(* Logix 5000 project; controller BTS01 vendor 1 type 14 code 217 rev 32.14; software revision 32.04; part 8 of 15 *)
(* tags used below, declared in another part *)
   Alarm_Active : DINT;
   Alarm_TMR : TIMER[17,32];
   ALM_ENABLE : DINT[25];
   HMI_Global_Alarm_Ack_PB : BOOL;
   HMIAlarms : DINT[25];   // Alarm Trigger Array
   HMIAlarmsMsg : STRING64[17,32];   // Alarm Descriptions to Match Alarm Trigger Array
(* Alarm, continued *)

ROUTINE Alarm_07   (* ladder *)
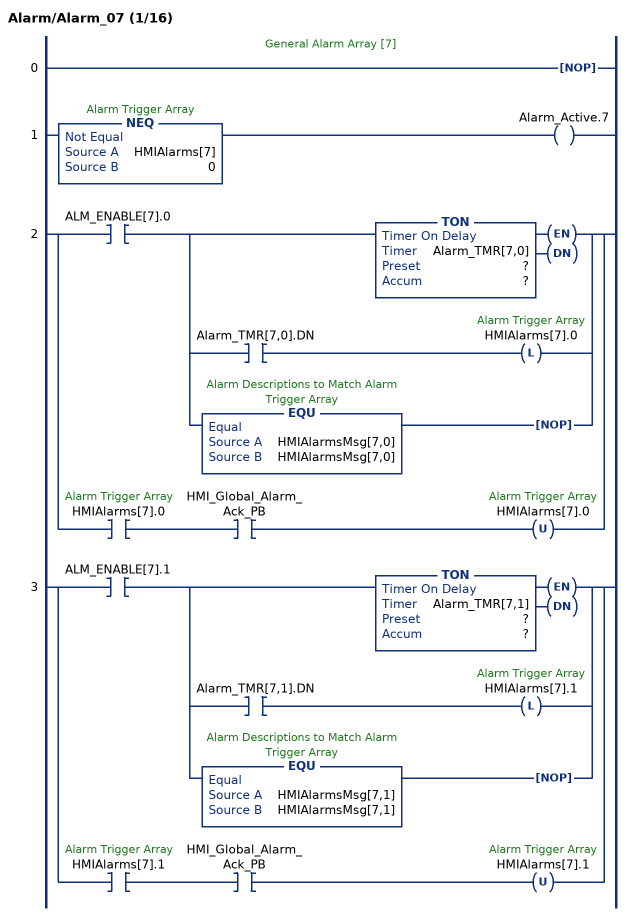
   // General Alarm Array [7]
   0: NOP();
   1: NEQ(HMIAlarms[7],0)OTE(Alarm_Active.7);
   2: [XIC(ALM_ENABLE[7].0) [TON(Alarm_TMR[7,0],?,?) ,XIC(Alarm_TMR[7,0].DN) OTL(HMIAlarms[7].0) ,EQU(HMIAlarmsMsg[7,0],HMIAlarmsMsg[7,0]) NOP() ] ,XIC(HMIAlarms[7].0) XIC(HMI_Global_Alarm_Ack_PB) OTU(HMIAlarms[7].0) ];
   3: [XIC(ALM_ENABLE[7].1) [TON(Alarm_TMR[7,1],?,?) ,XIC(Alarm_TMR[7,1].DN) OTL(HMIAlarms[7].1) ,EQU(HMIAlarmsMsg[7,1],HMIAlarmsMsg[7,1]) NOP() ] ,XIC(HMIAlarms[7].1) XIC(HMI_Global_Alarm_Ack_PB) OTU(HMIAlarms[7].1) ];
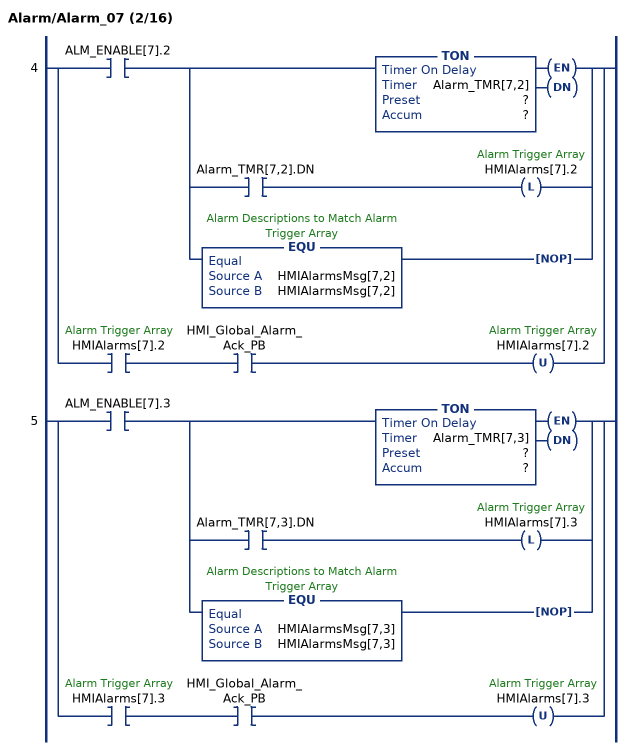
   4: [XIC(ALM_ENABLE[7].2) [TON(Alarm_TMR[7,2],?,?) ,XIC(Alarm_TMR[7,2].DN) OTL(HMIAlarms[7].2) ,EQU(HMIAlarmsMsg[7,2],HMIAlarmsMsg[7,2]) NOP() ] ,XIC(HMIAlarms[7].2) XIC(HMI_Global_Alarm_Ack_PB) OTU(HMIAlarms[7].2) ];
   5: [XIC(ALM_ENABLE[7].3) [TON(Alarm_TMR[7,3],?,?) ,XIC(Alarm_TMR[7,3].DN) OTL(HMIAlarms[7].3) ,EQU(HMIAlarmsMsg[7,3],HMIAlarmsMsg[7,3]) NOP() ] ,XIC(HMIAlarms[7].3) XIC(HMI_Global_Alarm_Ack_PB) OTU(HMIAlarms[7].3) ];
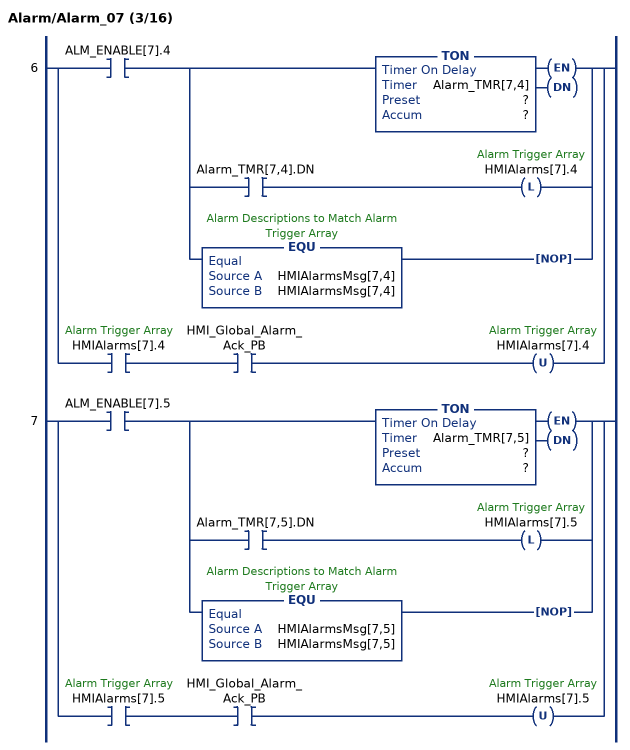
   6: [XIC(ALM_ENABLE[7].4) [TON(Alarm_TMR[7,4],?,?) ,XIC(Alarm_TMR[7,4].DN) OTL(HMIAlarms[7].4) ,EQU(HMIAlarmsMsg[7,4],HMIAlarmsMsg[7,4]) NOP() ] ,XIC(HMIAlarms[7].4) XIC(HMI_Global_Alarm_Ack_PB) OTU(HMIAlarms[7].4) ];
   7: [XIC(ALM_ENABLE[7].5) [TON(Alarm_TMR[7,5],?,?) ,XIC(Alarm_TMR[7,5].DN) OTL(HMIAlarms[7].5) ,EQU(HMIAlarmsMsg[7,5],HMIAlarmsMsg[7,5]) NOP() ] ,XIC(HMIAlarms[7].5) XIC(HMI_Global_Alarm_Ack_PB) OTU(HMIAlarms[7].5) ];
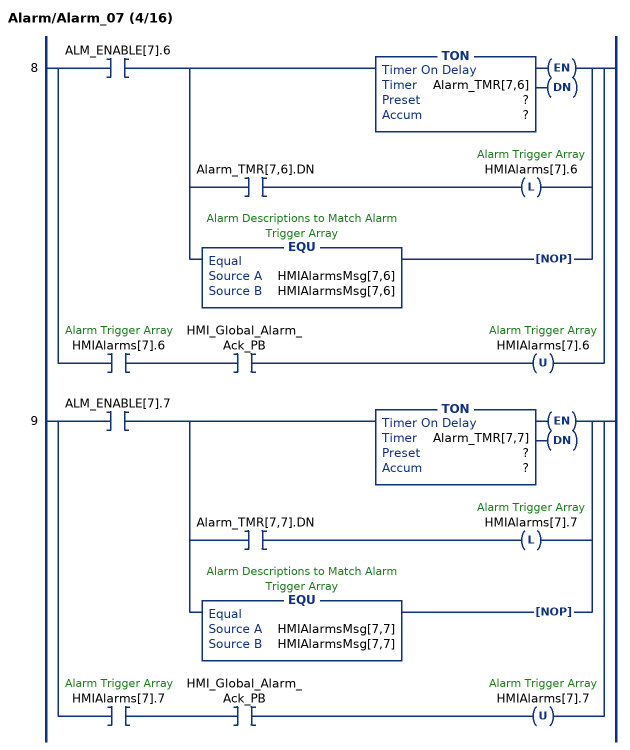
   8: [XIC(ALM_ENABLE[7].6) [TON(Alarm_TMR[7,6],?,?) ,XIC(Alarm_TMR[7,6].DN) OTL(HMIAlarms[7].6) ,EQU(HMIAlarmsMsg[7,6],HMIAlarmsMsg[7,6]) NOP() ] ,XIC(HMIAlarms[7].6) XIC(HMI_Global_Alarm_Ack_PB) OTU(HMIAlarms[7].6) ];
   9: [XIC(ALM_ENABLE[7].7) [TON(Alarm_TMR[7,7],?,?) ,XIC(Alarm_TMR[7,7].DN) OTL(HMIAlarms[7].7) ,EQU(HMIAlarmsMsg[7,7],HMIAlarmsMsg[7,7]) NOP() ] ,XIC(HMIAlarms[7].7) XIC(HMI_Global_Alarm_Ack_PB) OTU(HMIAlarms[7].7) ];
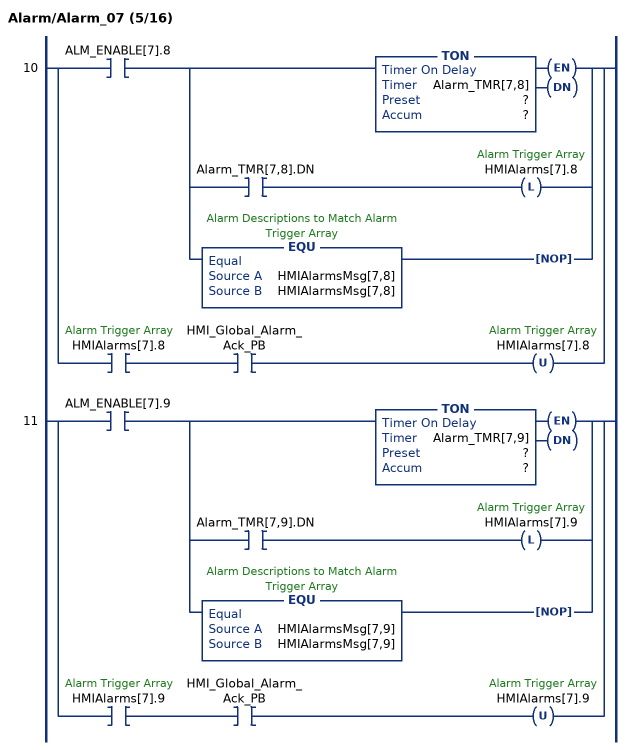
   10: [XIC(ALM_ENABLE[7].8) [TON(Alarm_TMR[7,8],?,?) ,XIC(Alarm_TMR[7,8].DN) OTL(HMIAlarms[7].8) ,EQU(HMIAlarmsMsg[7,8],HMIAlarmsMsg[7,8]) NOP() ] ,XIC(HMIAlarms[7].8) XIC(HMI_Global_Alarm_Ack_PB) OTU(HMIAlarms[7].8) ];
   11: [XIC(ALM_ENABLE[7].9) [TON(Alarm_TMR[7,9],?,?) ,XIC(Alarm_TMR[7,9].DN) OTL(HMIAlarms[7].9) ,EQU(HMIAlarmsMsg[7,9],HMIAlarmsMsg[7,9]) NOP() ] ,XIC(HMIAlarms[7].9) XIC(HMI_Global_Alarm_Ack_PB) OTU(HMIAlarms[7].9) ];
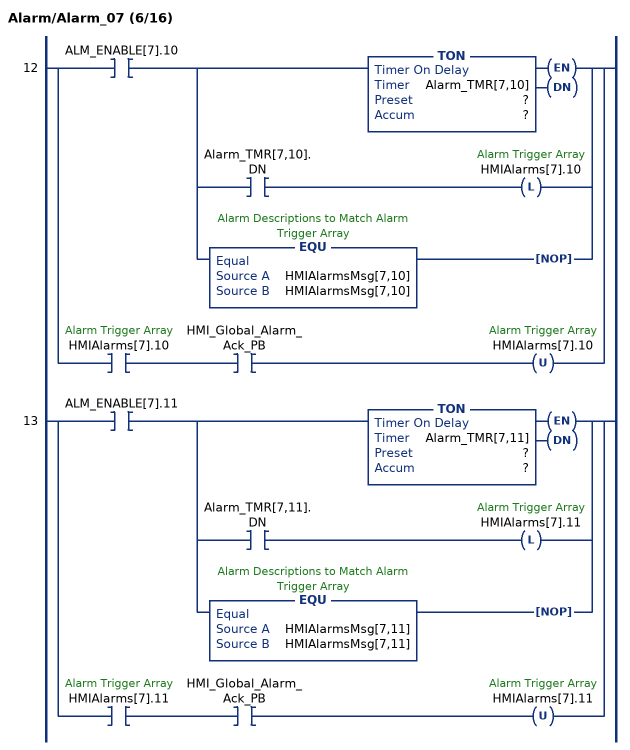
   12: [XIC(ALM_ENABLE[7].10) [TON(Alarm_TMR[7,10],?,?) ,XIC(Alarm_TMR[7,10].DN) OTL(HMIAlarms[7].10) ,EQU(HMIAlarmsMsg[7,10],HMIAlarmsMsg[7,10]) NOP() ] ,XIC(HMIAlarms[7].10) XIC(HMI_Global_Alarm_Ack_PB) OTU(HMIAlarms[7].10) ];
   13: [XIC(ALM_ENABLE[7].11) [TON(Alarm_TMR[7,11],?,?) ,XIC(Alarm_TMR[7,11].DN) OTL(HMIAlarms[7].11) ,EQU(HMIAlarmsMsg[7,11],HMIAlarmsMsg[7,11]) NOP() ] ,XIC(HMIAlarms[7].11) XIC(HMI_Global_Alarm_Ack_PB) OTU(HMIAlarms[7].11) ];
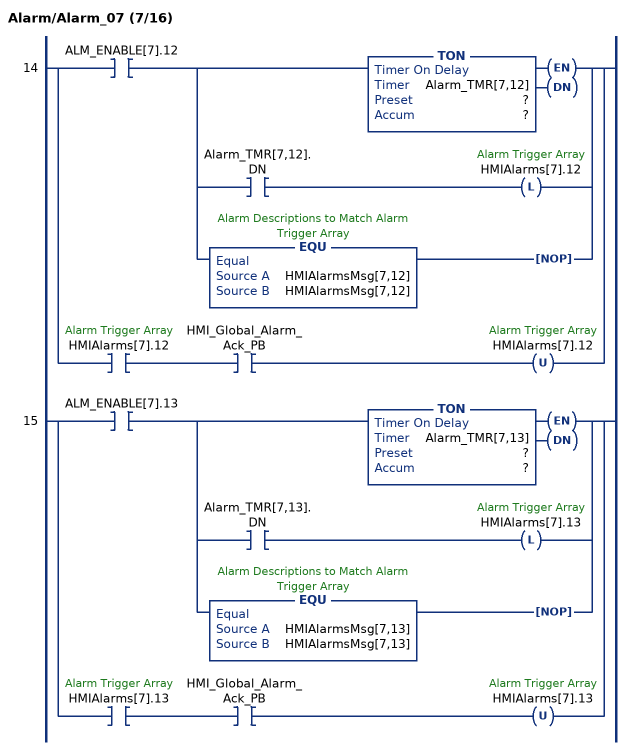
   14: [XIC(ALM_ENABLE[7].12) [TON(Alarm_TMR[7,12],?,?) ,XIC(Alarm_TMR[7,12].DN) OTL(HMIAlarms[7].12) ,EQU(HMIAlarmsMsg[7,12],HMIAlarmsMsg[7,12]) NOP() ] ,XIC(HMIAlarms[7].12) XIC(HMI_Global_Alarm_Ack_PB) OTU(HMIAlarms[7].12) ];
   15: [XIC(ALM_ENABLE[7].13) [TON(Alarm_TMR[7,13],?,?) ,XIC(Alarm_TMR[7,13].DN) OTL(HMIAlarms[7].13) ,EQU(HMIAlarmsMsg[7,13],HMIAlarmsMsg[7,13]) NOP() ] ,XIC(HMIAlarms[7].13) XIC(HMI_Global_Alarm_Ack_PB) OTU(HMIAlarms[7].13) ];
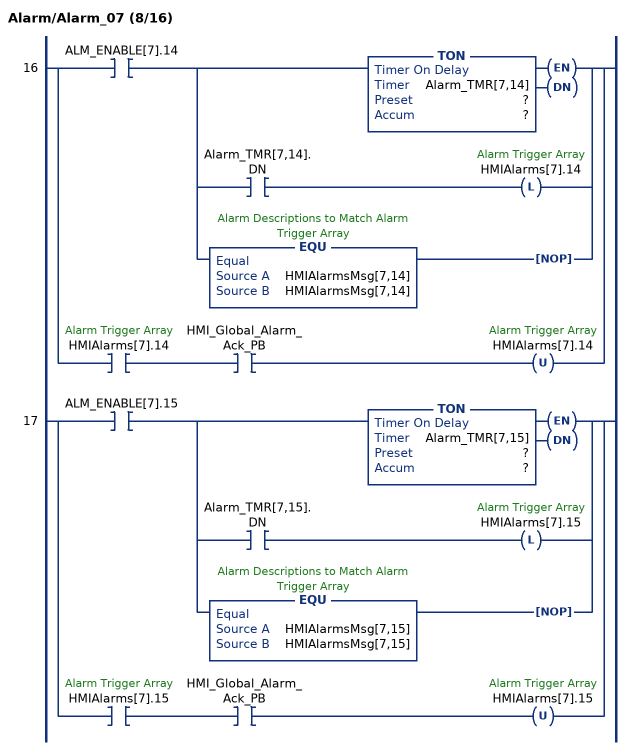
   16: [XIC(ALM_ENABLE[7].14) [TON(Alarm_TMR[7,14],?,?) ,XIC(Alarm_TMR[7,14].DN) OTL(HMIAlarms[7].14) ,EQU(HMIAlarmsMsg[7,14],HMIAlarmsMsg[7,14]) NOP() ] ,XIC(HMIAlarms[7].14) XIC(HMI_Global_Alarm_Ack_PB) OTU(HMIAlarms[7].14) ];
   17: [XIC(ALM_ENABLE[7].15) [TON(Alarm_TMR[7,15],?,?) ,XIC(Alarm_TMR[7,15].DN) OTL(HMIAlarms[7].15) ,EQU(HMIAlarmsMsg[7,15],HMIAlarmsMsg[7,15]) NOP() ] ,XIC(HMIAlarms[7].15) XIC(HMI_Global_Alarm_Ack_PB) OTU(HMIAlarms[7].15) ];
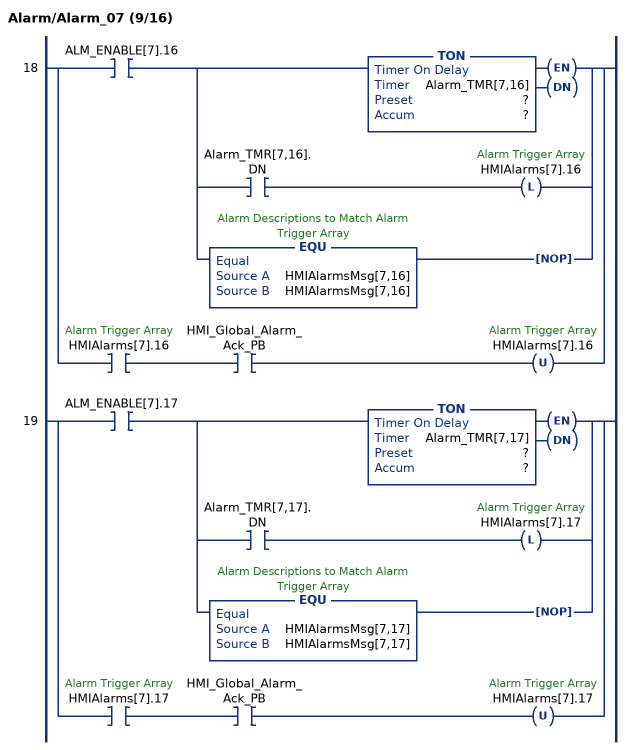
   18: [XIC(ALM_ENABLE[7].16) [TON(Alarm_TMR[7,16],?,?) ,XIC(Alarm_TMR[7,16].DN) OTL(HMIAlarms[7].16) ,EQU(HMIAlarmsMsg[7,16],HMIAlarmsMsg[7,16]) NOP() ] ,XIC(HMIAlarms[7].16) XIC(HMI_Global_Alarm_Ack_PB) OTU(HMIAlarms[7].16) ];
   19: [XIC(ALM_ENABLE[7].17) [TON(Alarm_TMR[7,17],?,?) ,XIC(Alarm_TMR[7,17].DN) OTL(HMIAlarms[7].17) ,EQU(HMIAlarmsMsg[7,17],HMIAlarmsMsg[7,17]) NOP() ] ,XIC(HMIAlarms[7].17) XIC(HMI_Global_Alarm_Ack_PB) OTU(HMIAlarms[7].17) ];
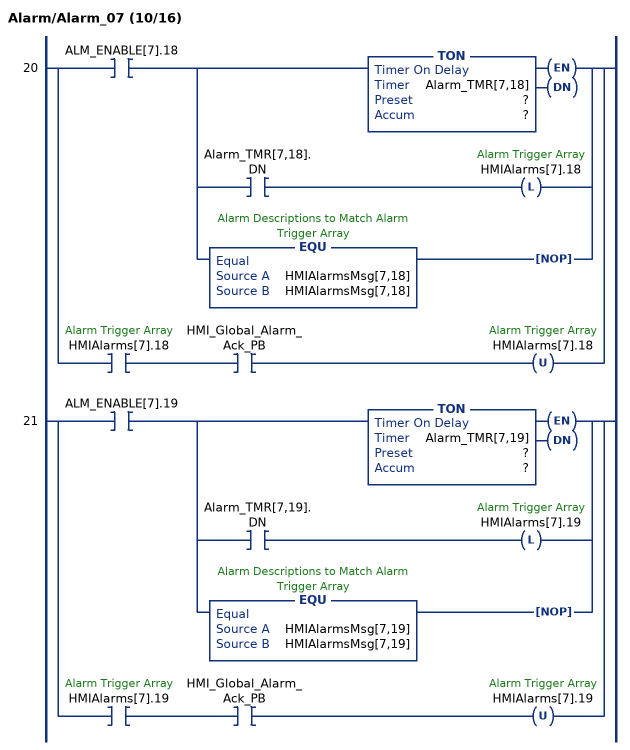
   20: [XIC(ALM_ENABLE[7].18) [TON(Alarm_TMR[7,18],?,?) ,XIC(Alarm_TMR[7,18].DN) OTL(HMIAlarms[7].18) ,EQU(HMIAlarmsMsg[7,18],HMIAlarmsMsg[7,18]) NOP() ] ,XIC(HMIAlarms[7].18) XIC(HMI_Global_Alarm_Ack_PB) OTU(HMIAlarms[7].18) ];
   21: [XIC(ALM_ENABLE[7].19) [TON(Alarm_TMR[7,19],?,?) ,XIC(Alarm_TMR[7,19].DN) OTL(HMIAlarms[7].19) ,EQU(HMIAlarmsMsg[7,19],HMIAlarmsMsg[7,19]) NOP() ] ,XIC(HMIAlarms[7].19) XIC(HMI_Global_Alarm_Ack_PB) OTU(HMIAlarms[7].19) ];
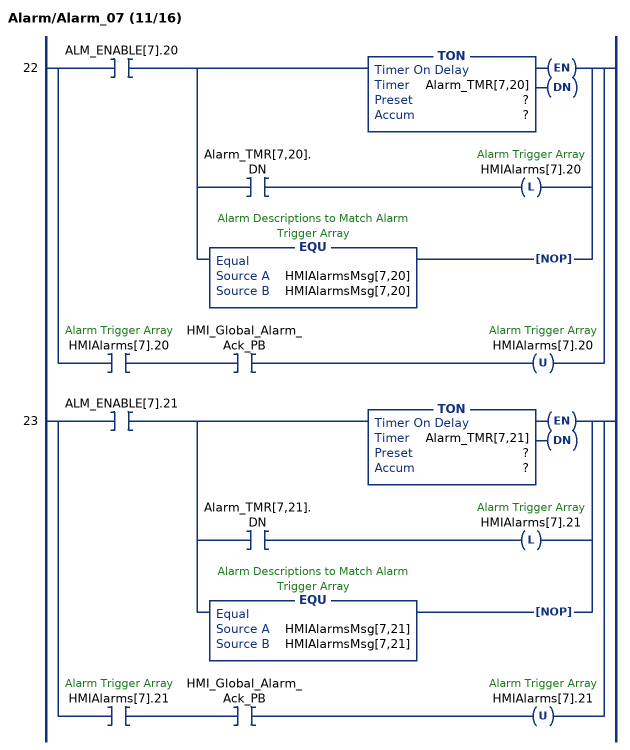
   22: [XIC(ALM_ENABLE[7].20) [TON(Alarm_TMR[7,20],?,?) ,XIC(Alarm_TMR[7,20].DN) OTL(HMIAlarms[7].20) ,EQU(HMIAlarmsMsg[7,20],HMIAlarmsMsg[7,20]) NOP() ] ,XIC(HMIAlarms[7].20) XIC(HMI_Global_Alarm_Ack_PB) OTU(HMIAlarms[7].20) ];
   23: [XIC(ALM_ENABLE[7].21) [TON(Alarm_TMR[7,21],?,?) ,XIC(Alarm_TMR[7,21].DN) OTL(HMIAlarms[7].21) ,EQU(HMIAlarmsMsg[7,21],HMIAlarmsMsg[7,21]) NOP() ] ,XIC(HMIAlarms[7].21) XIC(HMI_Global_Alarm_Ack_PB) OTU(HMIAlarms[7].21) ];
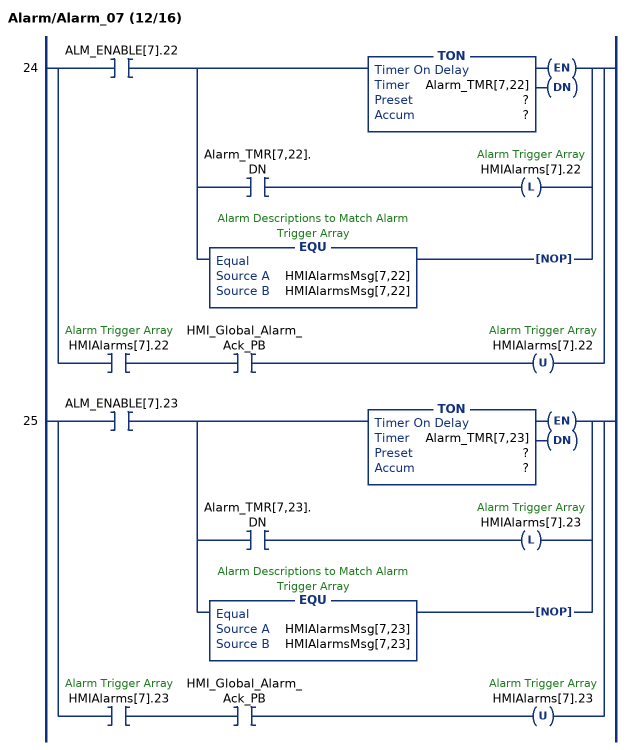
   24: [XIC(ALM_ENABLE[7].22) [TON(Alarm_TMR[7,22],?,?) ,XIC(Alarm_TMR[7,22].DN) OTL(HMIAlarms[7].22) ,EQU(HMIAlarmsMsg[7,22],HMIAlarmsMsg[7,22]) NOP() ] ,XIC(HMIAlarms[7].22) XIC(HMI_Global_Alarm_Ack_PB) OTU(HMIAlarms[7].22) ];
   25: [XIC(ALM_ENABLE[7].23) [TON(Alarm_TMR[7,23],?,?) ,XIC(Alarm_TMR[7,23].DN) OTL(HMIAlarms[7].23) ,EQU(HMIAlarmsMsg[7,23],HMIAlarmsMsg[7,23]) NOP() ] ,XIC(HMIAlarms[7].23) XIC(HMI_Global_Alarm_Ack_PB) OTU(HMIAlarms[7].23) ];
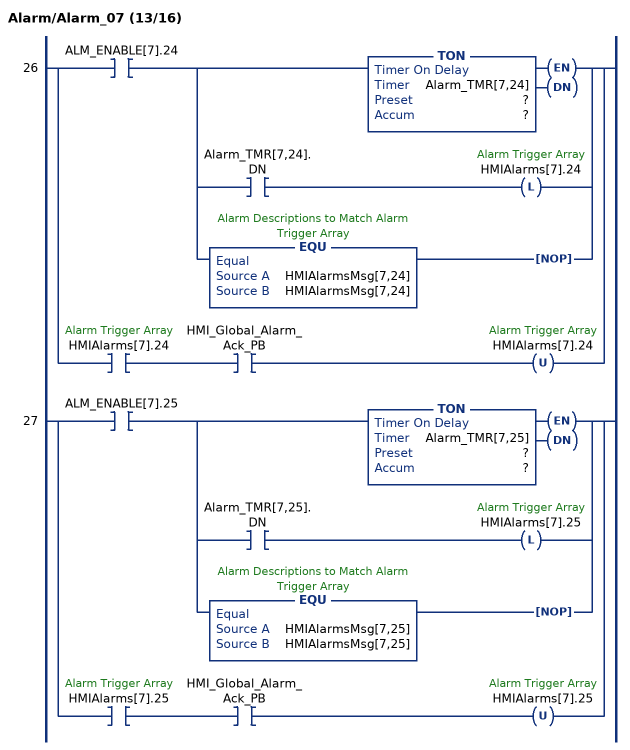
   26: [XIC(ALM_ENABLE[7].24) [TON(Alarm_TMR[7,24],?,?) ,XIC(Alarm_TMR[7,24].DN) OTL(HMIAlarms[7].24) ,EQU(HMIAlarmsMsg[7,24],HMIAlarmsMsg[7,24]) NOP() ] ,XIC(HMIAlarms[7].24) XIC(HMI_Global_Alarm_Ack_PB) OTU(HMIAlarms[7].24) ];
   27: [XIC(ALM_ENABLE[7].25) [TON(Alarm_TMR[7,25],?,?) ,XIC(Alarm_TMR[7,25].DN) OTL(HMIAlarms[7].25) ,EQU(HMIAlarmsMsg[7,25],HMIAlarmsMsg[7,25]) NOP() ] ,XIC(HMIAlarms[7].25) XIC(HMI_Global_Alarm_Ack_PB) OTU(HMIAlarms[7].25) ];
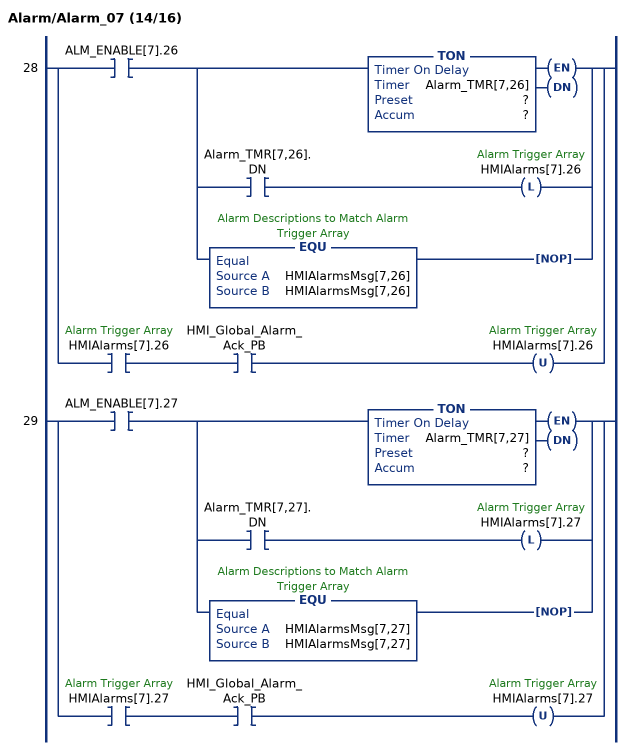
   28: [XIC(ALM_ENABLE[7].26) [TON(Alarm_TMR[7,26],?,?) ,XIC(Alarm_TMR[7,26].DN) OTL(HMIAlarms[7].26) ,EQU(HMIAlarmsMsg[7,26],HMIAlarmsMsg[7,26]) NOP() ] ,XIC(HMIAlarms[7].26) XIC(HMI_Global_Alarm_Ack_PB) OTU(HMIAlarms[7].26) ];
   29: [XIC(ALM_ENABLE[7].27) [TON(Alarm_TMR[7,27],?,?) ,XIC(Alarm_TMR[7,27].DN) OTL(HMIAlarms[7].27) ,EQU(HMIAlarmsMsg[7,27],HMIAlarmsMsg[7,27]) NOP() ] ,XIC(HMIAlarms[7].27) XIC(HMI_Global_Alarm_Ack_PB) OTU(HMIAlarms[7].27) ];
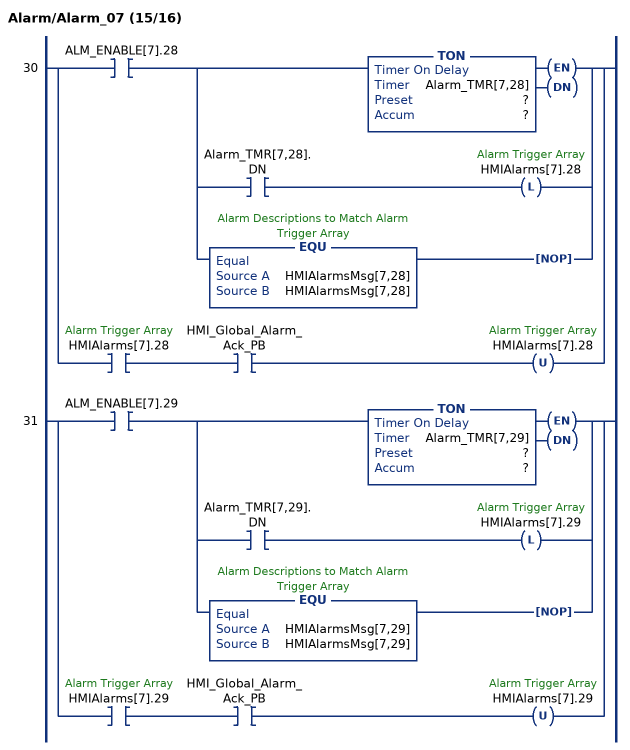
   30: [XIC(ALM_ENABLE[7].28) [TON(Alarm_TMR[7,28],?,?) ,XIC(Alarm_TMR[7,28].DN) OTL(HMIAlarms[7].28) ,EQU(HMIAlarmsMsg[7,28],HMIAlarmsMsg[7,28]) NOP() ] ,XIC(HMIAlarms[7].28) XIC(HMI_Global_Alarm_Ack_PB) OTU(HMIAlarms[7].28) ];
   31: [XIC(ALM_ENABLE[7].29) [TON(Alarm_TMR[7,29],?,?) ,XIC(Alarm_TMR[7,29].DN) OTL(HMIAlarms[7].29) ,EQU(HMIAlarmsMsg[7,29],HMIAlarmsMsg[7,29]) NOP() ] ,XIC(HMIAlarms[7].29) XIC(HMI_Global_Alarm_Ack_PB) OTU(HMIAlarms[7].29) ];
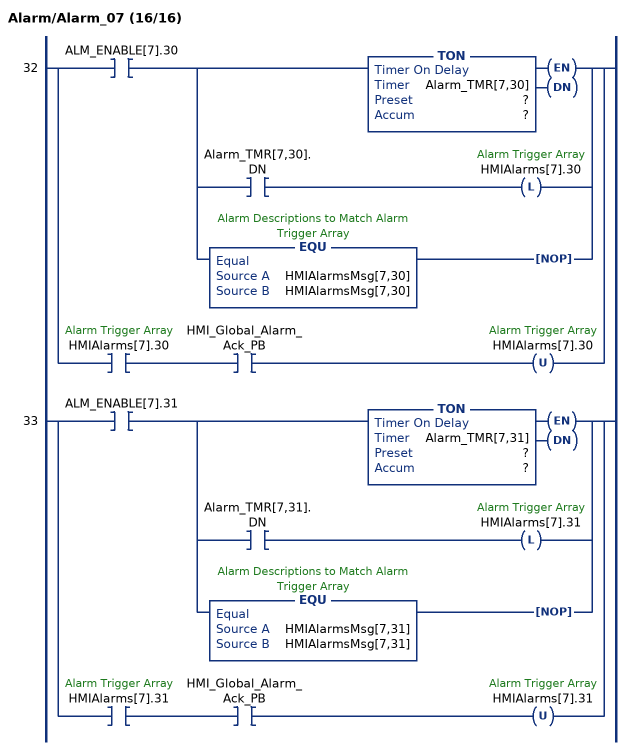
   32: [XIC(ALM_ENABLE[7].30) [TON(Alarm_TMR[7,30],?,?) ,XIC(Alarm_TMR[7,30].DN) OTL(HMIAlarms[7].30) ,EQU(HMIAlarmsMsg[7,30],HMIAlarmsMsg[7,30]) NOP() ] ,XIC(HMIAlarms[7].30) XIC(HMI_Global_Alarm_Ack_PB) OTU(HMIAlarms[7].30) ];
   33: [XIC(ALM_ENABLE[7].31) [TON(Alarm_TMR[7,31],?,?) ,XIC(Alarm_TMR[7,31].DN) OTL(HMIAlarms[7].31) ,EQU(HMIAlarmsMsg[7,31],HMIAlarmsMsg[7,31]) NOP() ] ,XIC(HMIAlarms[7].31) XIC(HMI_Global_Alarm_Ack_PB) OTU(HMIAlarms[7].31) ];
END_ROUTINE

ROUTINE Alarm_08   (* ladder *)
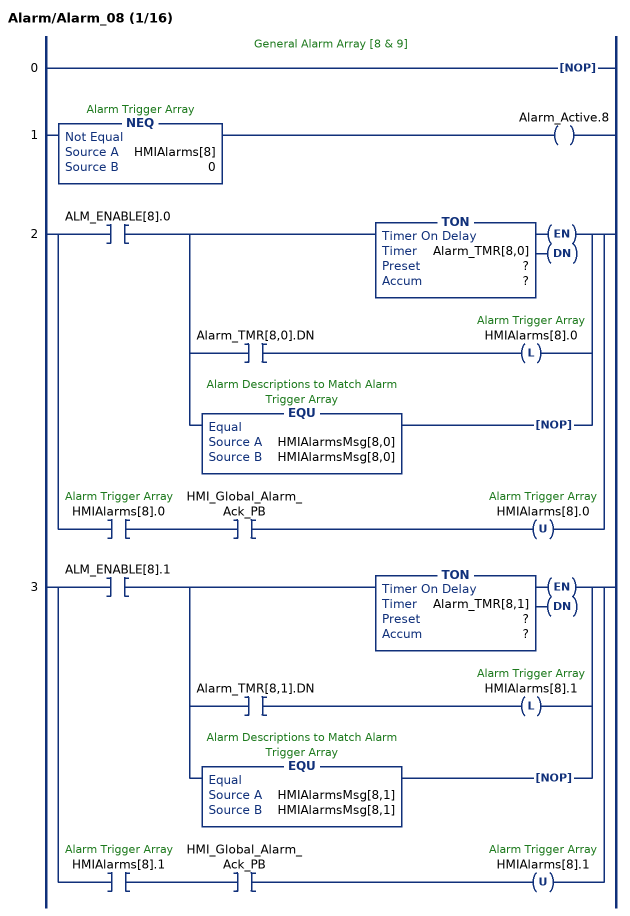
   // General Alarm Array [8 & 9]
   0: NOP();
   1: NEQ(HMIAlarms[8],0)OTE(Alarm_Active.8);
   2: [XIC(ALM_ENABLE[8].0) [TON(Alarm_TMR[8,0],?,?) ,XIC(Alarm_TMR[8,0].DN) OTL(HMIAlarms[8].0) ,EQU(HMIAlarmsMsg[8,0],HMIAlarmsMsg[8,0]) NOP() ] ,XIC(HMIAlarms[8].0) XIC(HMI_Global_Alarm_Ack_PB) OTU(HMIAlarms[8].0) ];
   3: [XIC(ALM_ENABLE[8].1) [TON(Alarm_TMR[8,1],?,?) ,XIC(Alarm_TMR[8,1].DN) OTL(HMIAlarms[8].1) ,EQU(HMIAlarmsMsg[8,1],HMIAlarmsMsg[8,1]) NOP() ] ,XIC(HMIAlarms[8].1) XIC(HMI_Global_Alarm_Ack_PB) OTU(HMIAlarms[8].1) ];
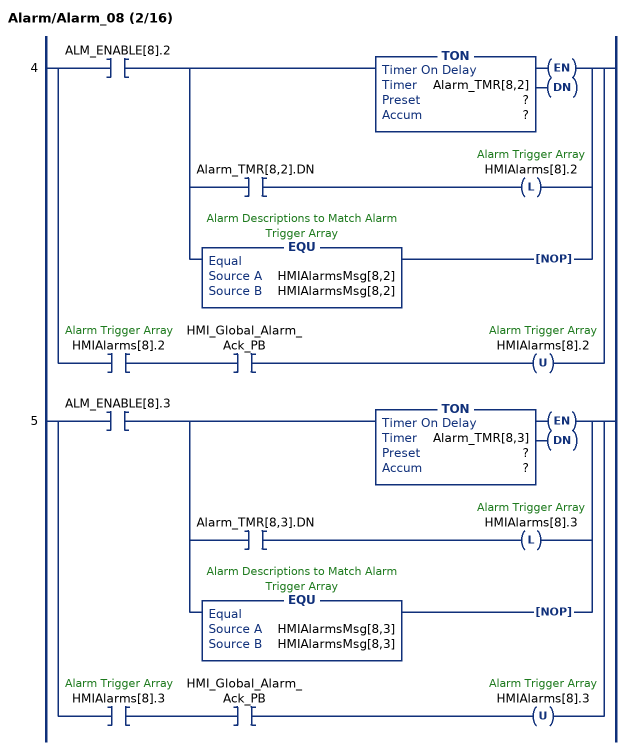
   4: [XIC(ALM_ENABLE[8].2) [TON(Alarm_TMR[8,2],?,?) ,XIC(Alarm_TMR[8,2].DN) OTL(HMIAlarms[8].2) ,EQU(HMIAlarmsMsg[8,2],HMIAlarmsMsg[8,2]) NOP() ] ,XIC(HMIAlarms[8].2) XIC(HMI_Global_Alarm_Ack_PB) OTU(HMIAlarms[8].2) ];
   5: [XIC(ALM_ENABLE[8].3) [TON(Alarm_TMR[8,3],?,?) ,XIC(Alarm_TMR[8,3].DN) OTL(HMIAlarms[8].3) ,EQU(HMIAlarmsMsg[8,3],HMIAlarmsMsg[8,3]) NOP() ] ,XIC(HMIAlarms[8].3) XIC(HMI_Global_Alarm_Ack_PB) OTU(HMIAlarms[8].3) ];
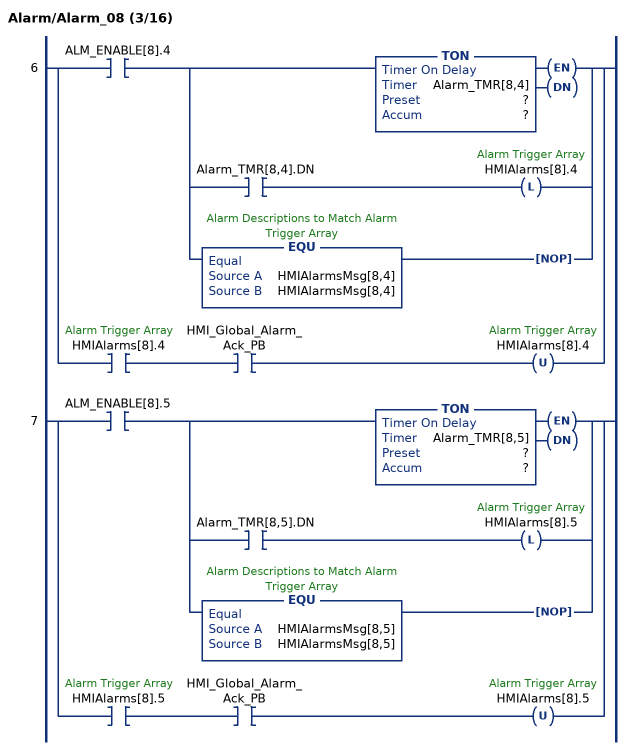
   6: [XIC(ALM_ENABLE[8].4) [TON(Alarm_TMR[8,4],?,?) ,XIC(Alarm_TMR[8,4].DN) OTL(HMIAlarms[8].4) ,EQU(HMIAlarmsMsg[8,4],HMIAlarmsMsg[8,4]) NOP() ] ,XIC(HMIAlarms[8].4) XIC(HMI_Global_Alarm_Ack_PB) OTU(HMIAlarms[8].4) ];
   7: [XIC(ALM_ENABLE[8].5) [TON(Alarm_TMR[8,5],?,?) ,XIC(Alarm_TMR[8,5].DN) OTL(HMIAlarms[8].5) ,EQU(HMIAlarmsMsg[8,5],HMIAlarmsMsg[8,5]) NOP() ] ,XIC(HMIAlarms[8].5) XIC(HMI_Global_Alarm_Ack_PB) OTU(HMIAlarms[8].5) ];
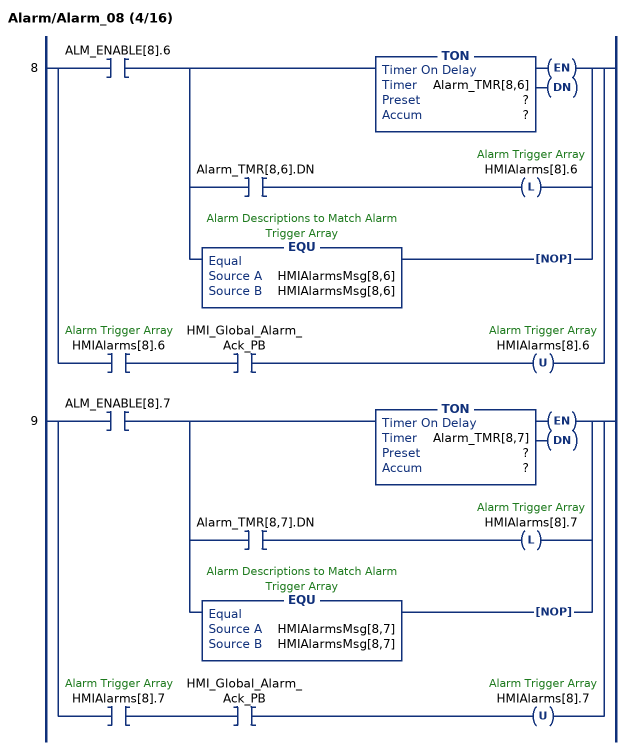
   8: [XIC(ALM_ENABLE[8].6) [TON(Alarm_TMR[8,6],?,?) ,XIC(Alarm_TMR[8,6].DN) OTL(HMIAlarms[8].6) ,EQU(HMIAlarmsMsg[8,6],HMIAlarmsMsg[8,6]) NOP() ] ,XIC(HMIAlarms[8].6) XIC(HMI_Global_Alarm_Ack_PB) OTU(HMIAlarms[8].6) ];
   9: [XIC(ALM_ENABLE[8].7) [TON(Alarm_TMR[8,7],?,?) ,XIC(Alarm_TMR[8,7].DN) OTL(HMIAlarms[8].7) ,EQU(HMIAlarmsMsg[8,7],HMIAlarmsMsg[8,7]) NOP() ] ,XIC(HMIAlarms[8].7) XIC(HMI_Global_Alarm_Ack_PB) OTU(HMIAlarms[8].7) ];
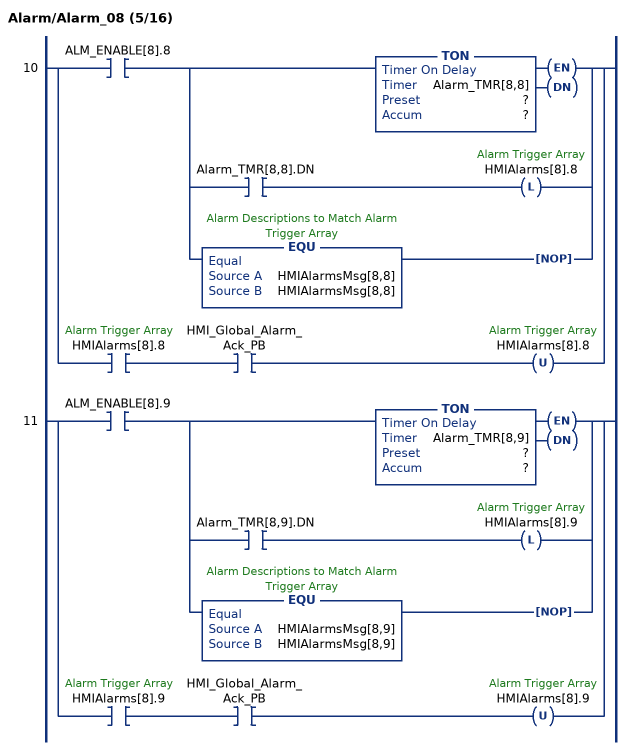
   10: [XIC(ALM_ENABLE[8].8) [TON(Alarm_TMR[8,8],?,?) ,XIC(Alarm_TMR[8,8].DN) OTL(HMIAlarms[8].8) ,EQU(HMIAlarmsMsg[8,8],HMIAlarmsMsg[8,8]) NOP() ] ,XIC(HMIAlarms[8].8) XIC(HMI_Global_Alarm_Ack_PB) OTU(HMIAlarms[8].8) ];
   11: [XIC(ALM_ENABLE[8].9) [TON(Alarm_TMR[8,9],?,?) ,XIC(Alarm_TMR[8,9].DN) OTL(HMIAlarms[8].9) ,EQU(HMIAlarmsMsg[8,9],HMIAlarmsMsg[8,9]) NOP() ] ,XIC(HMIAlarms[8].9) XIC(HMI_Global_Alarm_Ack_PB) OTU(HMIAlarms[8].9) ];
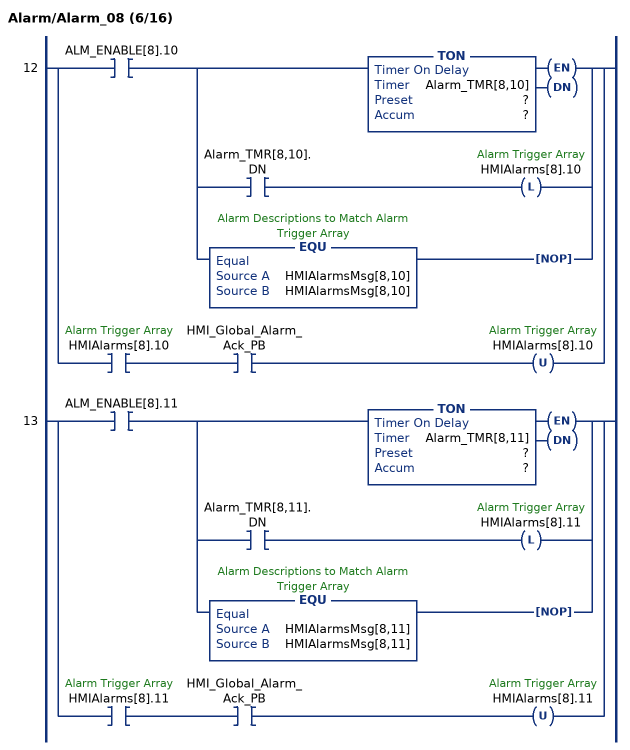
   12: [XIC(ALM_ENABLE[8].10) [TON(Alarm_TMR[8,10],?,?) ,XIC(Alarm_TMR[8,10].DN) OTL(HMIAlarms[8].10) ,EQU(HMIAlarmsMsg[8,10],HMIAlarmsMsg[8,10]) NOP() ] ,XIC(HMIAlarms[8].10) XIC(HMI_Global_Alarm_Ack_PB) OTU(HMIAlarms[8].10) ];
   13: [XIC(ALM_ENABLE[8].11) [TON(Alarm_TMR[8,11],?,?) ,XIC(Alarm_TMR[8,11].DN) OTL(HMIAlarms[8].11) ,EQU(HMIAlarmsMsg[8,11],HMIAlarmsMsg[8,11]) NOP() ] ,XIC(HMIAlarms[8].11) XIC(HMI_Global_Alarm_Ack_PB) OTU(HMIAlarms[8].11) ];
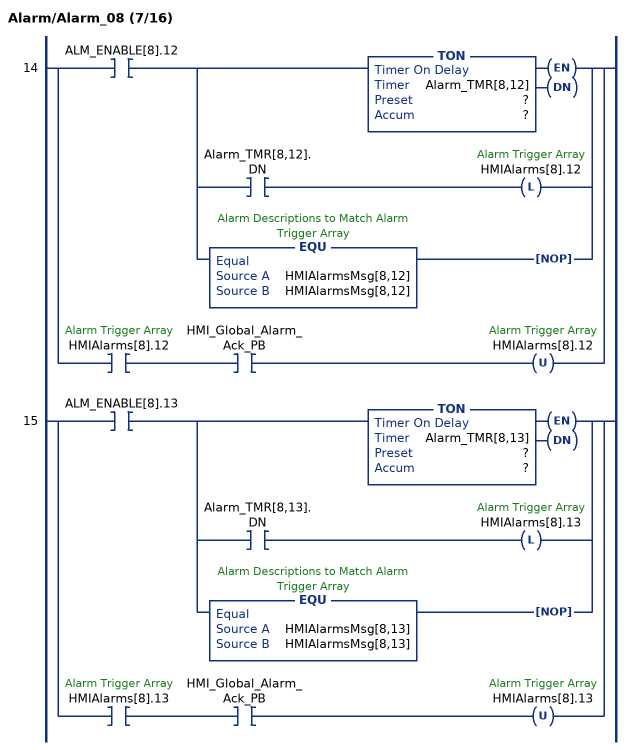
   14: [XIC(ALM_ENABLE[8].12) [TON(Alarm_TMR[8,12],?,?) ,XIC(Alarm_TMR[8,12].DN) OTL(HMIAlarms[8].12) ,EQU(HMIAlarmsMsg[8,12],HMIAlarmsMsg[8,12]) NOP() ] ,XIC(HMIAlarms[8].12) XIC(HMI_Global_Alarm_Ack_PB) OTU(HMIAlarms[8].12) ];
   15: [XIC(ALM_ENABLE[8].13) [TON(Alarm_TMR[8,13],?,?) ,XIC(Alarm_TMR[8,13].DN) OTL(HMIAlarms[8].13) ,EQU(HMIAlarmsMsg[8,13],HMIAlarmsMsg[8,13]) NOP() ] ,XIC(HMIAlarms[8].13) XIC(HMI_Global_Alarm_Ack_PB) OTU(HMIAlarms[8].13) ];
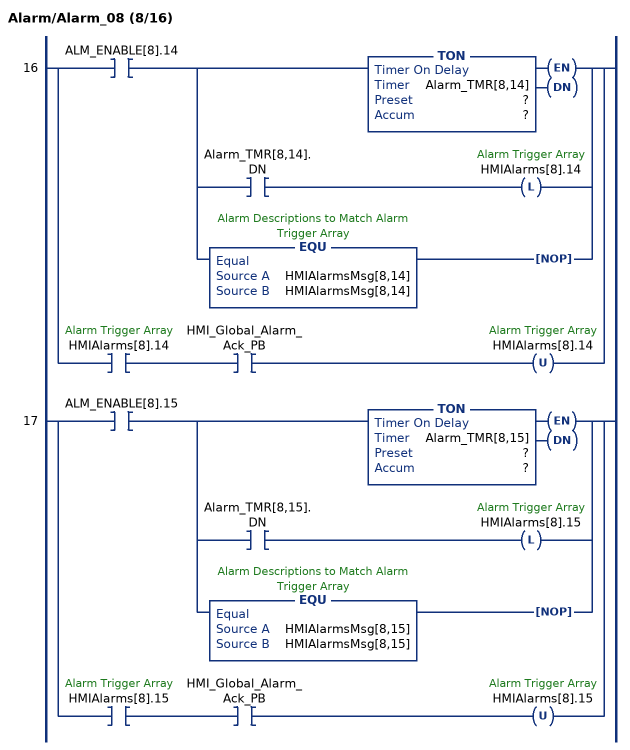
   16: [XIC(ALM_ENABLE[8].14) [TON(Alarm_TMR[8,14],?,?) ,XIC(Alarm_TMR[8,14].DN) OTL(HMIAlarms[8].14) ,EQU(HMIAlarmsMsg[8,14],HMIAlarmsMsg[8,14]) NOP() ] ,XIC(HMIAlarms[8].14) XIC(HMI_Global_Alarm_Ack_PB) OTU(HMIAlarms[8].14) ];
   17: [XIC(ALM_ENABLE[8].15) [TON(Alarm_TMR[8,15],?,?) ,XIC(Alarm_TMR[8,15].DN) OTL(HMIAlarms[8].15) ,EQU(HMIAlarmsMsg[8,15],HMIAlarmsMsg[8,15]) NOP() ] ,XIC(HMIAlarms[8].15) XIC(HMI_Global_Alarm_Ack_PB) OTU(HMIAlarms[8].15) ];
